(* Logix 5000 project; controller Lab1 vendor 1 type 14 code 155 rev 20.12; software revision 20.01 *)

TASK MainTask (continuous, watchdog 500 ms) : MainProgram

MODULES
   Local : vendor 1 type 14 code 155 (PointIO 0, rev 20.12)
      A_In : 1734-IE2V (PointIO 2, rev 3.1, Input RPI 80 ms)
      Stepper_1 : vendor 10 type 150 code 185 (PointIO 5, rev 1.1, Output RPI 50 ms)
      Stepper_2 : vendor 10 type 150 code 185 (PointIO 6, rev 1.1, Output RPI 50 ms)
      Discrete_IO : Embedded (PointIO 1, rev 20.11, Output RPI 20 ms)
      A_Out : 1734-OE2V (PointIO 3, rev 3.1, Output RPI 80 ms)
      HSC : vendor 1 type 109 code 13 (PointIO 4, rev 3.1, Output RPI 80 ms)
END_MODULES

PROGRAM MainProgram   (* main routine MainRoutine *)
VAR
   OUTPUT : DINT := 96;
   REVERSE : BOOL;
   STATE : INT;
   Stepper_Position : COUNTER := (PRE := 100, DN := 1);
   Stepper_Timer : TIMER := (PRE := 80, EN := 1, DN := 1);
END_VAR

ROUTINE MainRoutine   (* ladder *)
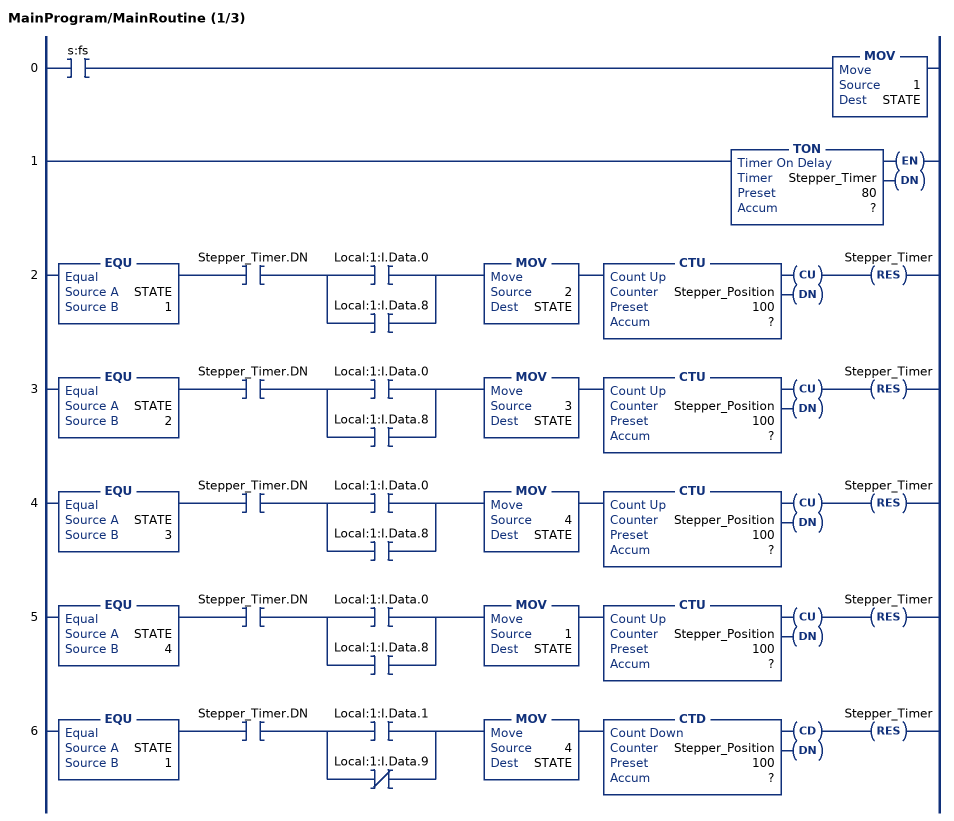
   0: XIC(s:fs)MOV(1,STATE);
   1: TON(Stepper_Timer,?,?);
   2: EQU(STATE,1)XIC(Stepper_Timer.DN)[XIC(Local:1:I.Data.0) ,XIC(Local:1:I.Data.8) ]MOV(2,STATE)CTU(Stepper_Position,?,?)RES(Stepper_Timer);
   3: EQU(STATE,2)XIC(Stepper_Timer.DN)[XIC(Local:1:I.Data.0) ,XIC(Local:1:I.Data.8) ]MOV(3,STATE)CTU(Stepper_Position,?,?)RES(Stepper_Timer);
   4: EQU(STATE,3)XIC(Stepper_Timer.DN)[XIC(Local:1:I.Data.0) ,XIC(Local:1:I.Data.8) ]MOV(4,STATE)CTU(Stepper_Position,?,?)RES(Stepper_Timer);
   5: EQU(STATE,4)XIC(Stepper_Timer.DN)[XIC(Local:1:I.Data.0) ,XIC(Local:1:I.Data.8) ]MOV(1,STATE)CTU(Stepper_Position,?,?)RES(Stepper_Timer);
   6: EQU(STATE,1)XIC(Stepper_Timer.DN)[XIC(Local:1:I.Data.1) ,XIO(Local:1:I.Data.9) ]MOV(4,STATE)CTD(Stepper_Position,?,?)RES(Stepper_Timer);
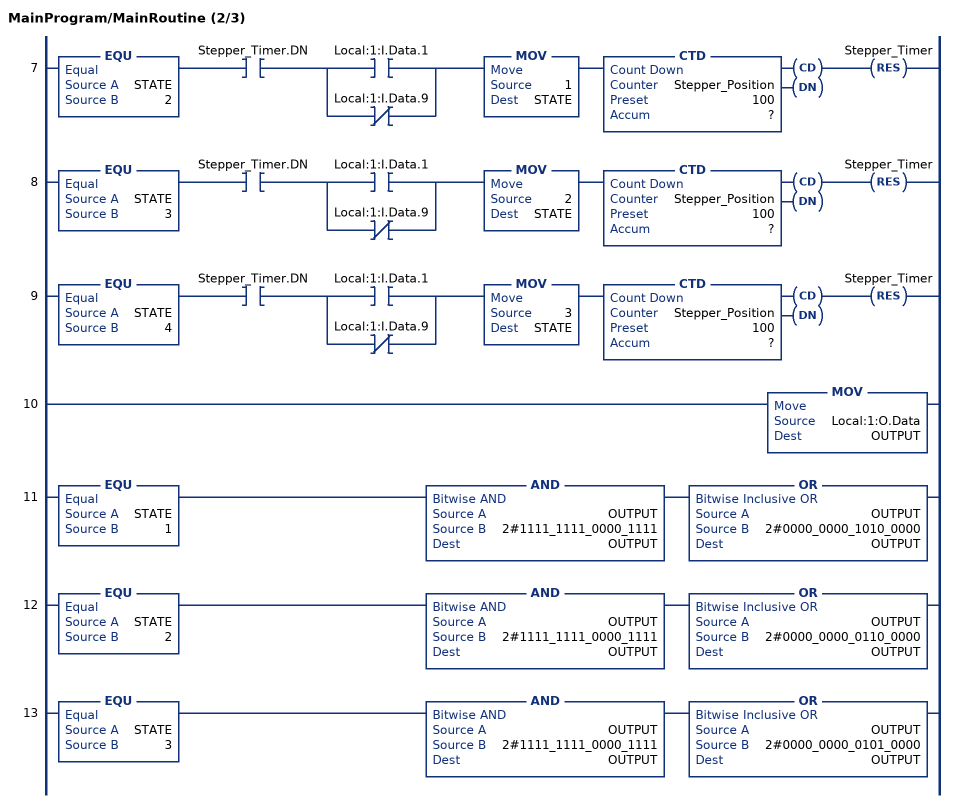
   7: EQU(STATE,2)XIC(Stepper_Timer.DN)[XIC(Local:1:I.Data.1) ,XIO(Local:1:I.Data.9) ]MOV(1,STATE)CTD(Stepper_Position,?,?)RES(Stepper_Timer);
   8: EQU(STATE,3)XIC(Stepper_Timer.DN)[XIC(Local:1:I.Data.1) ,XIO(Local:1:I.Data.9) ]MOV(2,STATE)CTD(Stepper_Position,?,?)RES(Stepper_Timer);
   9: EQU(STATE,4)XIC(Stepper_Timer.DN)[XIC(Local:1:I.Data.1) ,XIO(Local:1:I.Data.9) ]MOV(3,STATE)CTD(Stepper_Position,?,?)RES(Stepper_Timer);
   10: MOV(Local:1:O.Data,OUTPUT);
   11: EQU(STATE,1)AND(OUTPUT,2#1111_1111_0000_1111,OUTPUT)OR(OUTPUT,2#0000_0000_1010_0000,OUTPUT);
   12: EQU(STATE,2)AND(OUTPUT,2#1111_1111_0000_1111,OUTPUT)OR(OUTPUT,2#0000_0000_0110_0000,OUTPUT);
   13: EQU(STATE,3)AND(OUTPUT,2#1111_1111_0000_1111,OUTPUT)OR(OUTPUT,2#0000_0000_0101_0000,OUTPUT);
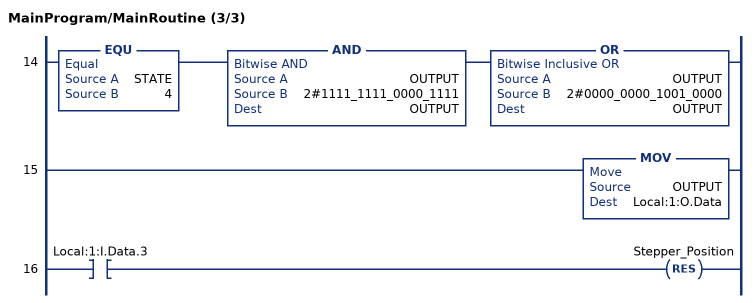
   14: EQU(STATE,4)AND(OUTPUT,2#1111_1111_0000_1111,OUTPUT)OR(OUTPUT,2#0000_0000_1001_0000,OUTPUT);
   15: MOV(OUTPUT,Local:1:O.Data);
   16: XIC(Local:1:I.Data.3)RES(Stepper_Position);
END_ROUTINE
END_PROGRAM
